Staubli VAL3: CartesianTrajPtMsg.dtx

public Header header
  [0]
    num nMsgType
    num nCommType
    num nReplyCode
    num nData[12]
public CartesianTrajPt cartesianTrajPt
  [0]
    num nSeq
    num nPosition[3]
    num nOrientation[4]
    num nVelocity
    num nAcceleration
    num nBlendingRadius
    num nDuration
public Prefix prefix
  [0]
    num nLength
    num nData[4]
public Body body
  [0]
    num nData[64]
